Staubli VAL3: find.pgx

public program find(string& x_sItem[] (dimensions=1), bool& x_bFound[] (dimensions=1))
begin
  // check if the item has been found
  x_bFound=isDefined(pt:tTraj[x_sItem])
end
